# EPICS autosave request: log/autosave/wcsIoc/wcsIoc.req
file wcsIoc0.req num=1
file wcsIoc0.req num=2
file wcsIoc0.req num=3
